// TIA Portal project "2022.06.06_标准与缩放指令" (V17)

(* hardware
DEVICE "S7-1200 station_1"  S7-1200 Station
   slot 0: "Rack_0"  S7-1200 Rack  Rack  V1.0
   slot 1: "PLC_1"  CPU 1212C DC/DC/DC  6ES7 212-1AE40-0XB0  V4.5
*)

// ===== PLC "PLC_1"  CPU 1212C DC/DC/DC =====

VAR_GLOBAL   // PLC tag table "默认变量表"
   "模拟量输入" AT %MW100 : Word;
   "Tag_3" AT %MW102 : UInt;
   "Tag_4" AT %MW104 : UInt;
   "Tag_5" AT %MW106 : UInt;
   "Tag_6" AT %I0.0 : Bool;
   "Tag_7" AT %M0.0 : Bool;
   "X(2)" AT %MW10 : Word;
   "Tag_9" AT %MW12 : UInt;
   "X" AT %MW0 : Word;
   "a" AT %MW2 : Word;
   "b" AT %MW4 : Int;
   "c" AT %MW8 : Int;
   "e" AT %MD0 : Real;
   "Tag_10" AT %MD2 : Real;
   "f" AT %MD4 : Real;
   "g" AT %MD8 : Real;
   "X(1)" AT %MD12 : Real;
   "Tag_8" AT %MD16 : Real;
   "中间值(1)" AT %MD200 : Real;
   "中间值" AT %MD104 : Real;
   "工程值" AT %MD108 : Real;
   "要求的频率" AT %MD60 : Real;
   "百分比" AT %MD64 : Real;
   "Tag_12" AT %MW70 : Int;
END_VAR

ORGANIZATION_BLOCK "Main"   // OB1, LAD, ProgramCycle
TITLE = "Main Program Sweep (Cycle)"
{ S7_Optimized_Access := 'TRUE' }
VERSION : 0.1
   VAR_INPUT
      Initial_Call : Bool;   // Initial call of this OB
      Remanence : Bool;   // =True, if remanent data are available
   END_VAR
BEGIN

REGION Network 1
   // 标准化：左边都是16进制，右边是浮点数。输出是小数，百分比
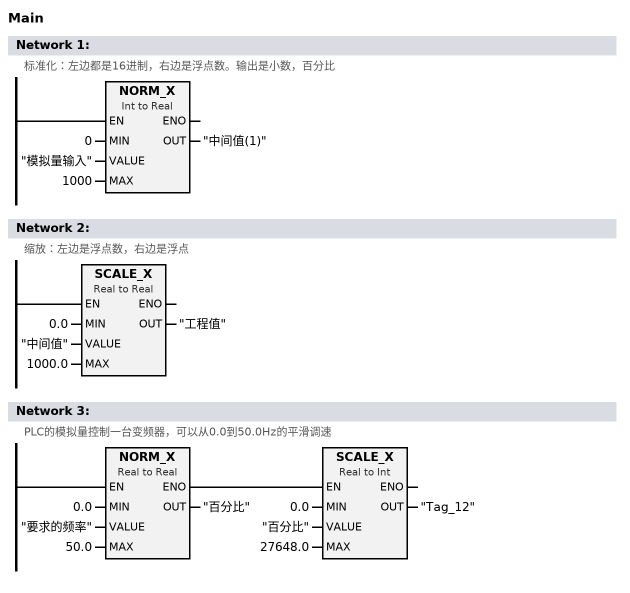
   RUNG wire#powerrail
      { S7_Templates := "[SrcType := Int, DestType := Real]" } Normalize(min := 0, value := "模拟量输入", max := 1000, out => "中间值(1)")
   END_RUNG
   // the same network as SCL:
   "中间值(1)" := NORM_X(MIN := 0, VALUE := "模拟量输入", MAX := 1000);
END_REGION

REGION Network 2
   // 缩放：左边是浮点数，右边是浮点
   RUNG wire#powerrail
      { S7_Templates := "[SrcType := Real, DestType := Real]" } Scale(min := 0.0, value := "中间值", max := 1000.0, out => "工程值")
   END_RUNG
   // the same network as SCL:
   "工程值" := SCALE_X(MIN := 0.0, VALUE := "中间值", MAX := 1000.0);
END_REGION

REGION Network 3
   // PLC的模拟量控制一台变频器，可以从0.0到50.0Hz的平滑调速
   RUNG wire#powerrail
      { S7_Templates := "[SrcType := Real, DestType := Real]" } Normalize(min := 0.0, value := "要求的频率", max := 50.0, out => "百分比")
      { S7_Templates := "[SrcType := Real, DestType := Int]" } Scale(min := 0.0, value := "百分比", max := 27648.0, out => "Tag_12")
   END_RUNG
   // the same network as SCL:
   "百分比" := NORM_X(MIN := 0.0, VALUE := "要求的频率", MAX := 50.0);
   "Tag_12" := SCALE_X(MIN := 0.0, VALUE := "百分比", MAX := 27648.0);
END_REGION
END_ORGANIZATION_BLOCK